(* Logix 5000 project; controller PlantaAutomatizacion vendor 1 type 14 code 156 rev 32.11; software revision 32.00 *)
// Planta de enesamblaje de patinetas electricas usando PLC Virtual.

TASK MainTask (continuous, watchdog 500 ms) : MainProgram

MODULES
   Local : vendor 1 type 14 code 156 (Compact 0, rev 32.11)
      Variador_141 : PowerFlex 525-EENET (Ethernet 10.203.3.141, rev 5.1, Output RPI 20 ms)
END_MODULES

VAR_GLOBAL   (* controller tags *)
   Banda1 : BOOL := 1;   // Motor de la banda 1
   Banda2 : BOOL := 1;   // Motor de la banda 2
   Banda3 : BOOL;   // Motor de la banda 3
   Banda4 : BOOL := 1;   // Motor de la Banda 4
   Banda5 : BOOL;   // Motor de la Banda 5
   Banda6 : BOOL;   // Motor de la banda 6
   Banda7 : BOOL;   // Motor de la Banda 7
   Google_Stp_Banda5 : BOOL;   // Stop con google assistant
   Google_Str_Banda5 : BOOL;   // Start Con Google Assistan
   RESET : BOOL;   // Reset del grafcet
   START : BOOL;   // Senal de inicio de la rutina
   StartBanda1 : BOOL := 1;   // Señal del sensor para activar Motor de la banda 1
   StartBanda2 : BOOL := 1;   // Señal del sensor para activar Motor de la banda 2
   StartBanda3 : BOOL;   // Señal del sensor para activar Motor de la banda 3
   StartBanda4 : BOOL := 1;   // Señal del sensor para activar Motor de la banda 4
   StartBanda5 : BOOL;   // Señal del sensor para activar Motor de la banda 5
   StartBanda6 : BOOL;   // Señal del sensor para activar Motor de la banda 6
   StartBanda7 : BOOL;   // Señal del sensor para activar Motor de la banda 7
   StopBanda1 : BOOL;   // Señal del sensor para desactivar Motor de la banda 1
   StopBanda2 : BOOL;   // Señal del sensor para desactivar Motor de la banda 2
   StopBanda3 : BOOL;   // Señal del sensor para desactivar Motor de la banda 3
   StopBanda4 : BOOL;   // Señal del sensor para desactivar Motor de la banda 4
   StopBanda5 : BOOL;   // Señal del sensor para desactivar Motor de la banda 5
   StopBanda6 : BOOL;   // Señal del sensor para desactivar Motor de la banda 6
   StopBanda7 : BOOL;   // Señal del sensor para desactivar Motor de la banda 7
END_VAR

PROGRAM MainProgram   (* main routine MainRoutine *)
VAR
   Action_000 : SFC_ACTION := (Status := 16#c020_0000, A := 1, Q := 1, PauseTimer := 1, Count := 1);   // Activar el Motor de la Banda
   Action_001 : SFC_ACTION := (Status := 16#0020_0000, PauseTimer := 1);
   Action_002 : SFC_ACTION := (Status := 16#c020_0000, A := 1, Q := 1, PauseTimer := 1, Count := 1);
   Action_003 : SFC_ACTION := (Status := 16#0020_0000, PauseTimer := 1);
   Action_004 : SFC_ACTION := (Status := 16#0020_0000, PauseTimer := 1);
   Action_005 : SFC_ACTION := (Status := 16#0020_0000, PauseTimer := 1);
   Action_006 : SFC_ACTION := (Status := 16#c020_0000, A := 1, Q := 1, PauseTimer := 1, Count := 1);
   Action_007 : SFC_ACTION := (Status := 16#0020_0000, PauseTimer := 1);
   Action_008 : SFC_ACTION := (Status := 16#0020_0000, PauseTimer := 1);
   Action_009 : SFC_ACTION := (Status := 16#0020_0000, PauseTimer := 1);
   Action_010 : SFC_ACTION := (Status := 16#0020_0000, PauseTimer := 1);
   Action_011 : SFC_ACTION := (Status := 16#0020_0000, PauseTimer := 1);
   Action_012 : SFC_ACTION := (Status := 16#0020_0000, PauseTimer := 1);
   Action_013 : SFC_ACTION := (Status := 16#0020_0000, PauseTimer := 1);
   Step_000 : SFC_STEP := (Status := 16#0820_0201, DN := 1, PauseTimer := 1, T := 400127, TMax := 400127, Count := 1);   // Paso Inicial
   Step_001 : SFC_STEP := (Status := 16#a820_0001, X := 1, SA := 1, DN := 1, PauseTimer := 1, T := 107426, TMax := 107426, Count := 1);   // Activar el Motor de la Banda
   Step_002 : SFC_STEP := (Status := 16#0020_0001, PauseTimer := 1);   // Detener el motor de la Banda
   Step_003 : SFC_STEP := (Status := 16#0820_0001, DN := 1, PauseTimer := 1, Count := 1);
   Step_004 : SFC_STEP := (Status := 16#a820_0001, X := 1, SA := 1, DN := 1, PauseTimer := 1, T := 107332, TMax := 107332, Count := 1);
   Step_005 : SFC_STEP := (Status := 16#0020_0001, PauseTimer := 1);
   Step_006 : SFC_STEP := (Status := 16#a820_0001, X := 1, SA := 1, DN := 1, PauseTimer := 1, T := 107361, TMax := 107361, Count := 1);
   Step_007 : SFC_STEP := (Status := 16#0020_0001, PauseTimer := 1);
   Step_008 : SFC_STEP := (Status := 16#0020_0001, PauseTimer := 1);
   Step_009 : SFC_STEP := (Status := 16#a820_0001, X := 1, SA := 1, DN := 1, PauseTimer := 1, T := 107408, TMax := 107408, Count := 1);
   Step_010 : SFC_STEP := (Status := 16#a820_0001, X := 1, SA := 1, DN := 1, PauseTimer := 1, T := 107437, TMax := 107437, Count := 1);
   Step_011 : SFC_STEP := (Status := 16#0020_0001, PauseTimer := 1);
   Step_012 : SFC_STEP := (Status := 16#a820_0001, X := 1, SA := 1, DN := 1, PauseTimer := 1, T := 107309, TMax := 107309, Count := 1);
   Step_013 : SFC_STEP := (Status := 16#0020_0001, PauseTimer := 1);
   Step_014 : SFC_STEP := (Status := 16#0020_0001, PauseTimer := 1);
   Step_015 : SFC_STEP := (Status := 16#0820_0001, DN := 1, PauseTimer := 1, Count := 1);   // Paso de paralelizado de las bandas
   Step_016 : SFC_STEP := (Status := 16#0020_0001, PauseTimer := 1);
   Step_017 : SFC_STEP := (Status := 16#0020_0001, PauseTimer := 1);
   Step_018 : SFC_STEP := (Status := 16#0820_0001, DN := 1, PauseTimer := 1, Count := 1);
   Step_019 : SFC_STEP := (Status := 16#a820_0001, X := 1, SA := 1, DN := 1, PauseTimer := 1, T := 107279, TMax := 107279, Count := 1);
   Step_020 : SFC_STEP := (Status := 16#0020_0001, PauseTimer := 1);
   Step_021 : SFC_STEP := (Status := 16#0020_0001, PauseTimer := 1);
   Tran_000 : BOOL := 1;   // Sensor de banda 1 indicando que hay un Objeto
   Tran_001 : BOOL;   // Sensor de parada, indicando qeu el objeto llego a su destino
   Tran_002 : BOOL;   // Cuando El objeto ya halla sido recogido Y otro objeto se encuentre al incio
   Tran_003 : BOOL := 1;
   Tran_004 : BOOL;
   Tran_005 : BOOL;
   Tran_006 : BOOL;
   Tran_007 : BOOL;
   Tran_008 : BOOL := 1;
   Tran_009 : BOOL := 1;
   Tran_010 : BOOL;
   Tran_011 : BOOL;
   Tran_012 : BOOL;
   Tran_013 : BOOL := 1;
   Tran_014 : BOOL;
   Tran_015 : BOOL;
   Tran_016 : BOOL := 1;
   Tran_017 : BOOL;
   Tran_018 : BOOL;
   Tran_019 : BOOL := 1;
   Tran_020 : BOOL;
   Tran_022 : BOOL := 1;   // START para empezar la logica grafcet
END_VAR

ROUTINE GrafcetBandas   (* sequential function chart *)
// Logica secuencial para el movimiento de las bandas
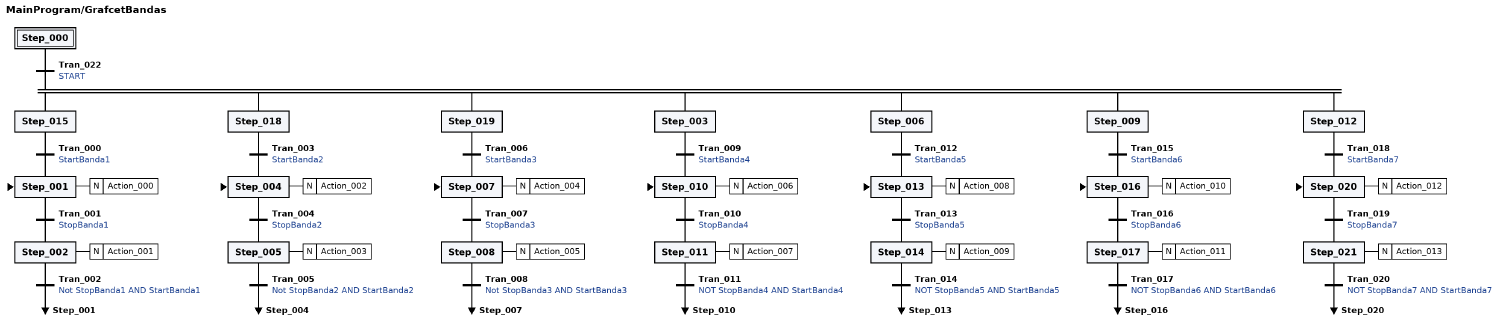
   // BANDA 1
   // BANDA 2
   // BANDA 3
   // BANDA 4
   // BANDA 5
   // BANDA 6
   // BANDA 7
   INITIAL_STEP Step_000:
   END_STEP
   TRANSITION Tran_022 FROM Step_000 TO (Step_018, Step_019, Step_015, Step_003, Step_006, Step_009, Step_012)
      := START
   END_TRANSITION
   STEP Step_015:
   END_STEP
   STEP Step_018:
   END_STEP
   STEP Step_019:
   END_STEP
   STEP Step_003:
   END_STEP
   STEP Step_006:
   END_STEP
   STEP Step_009:
   END_STEP
   STEP Step_012:
   END_STEP
   TRANSITION Tran_015 FROM Step_009 TO Step_016
      := StartBanda6
   END_TRANSITION
   TRANSITION Tran_018 FROM Step_012 TO Step_020
      := StartBanda7
   END_TRANSITION
   TRANSITION Tran_000 FROM Step_015 TO Step_001
      := StartBanda1
   END_TRANSITION
   TRANSITION Tran_003 FROM Step_018 TO Step_004
      := StartBanda2
   END_TRANSITION
   TRANSITION Tran_006 FROM Step_019 TO Step_007
      := StartBanda3
   END_TRANSITION
   TRANSITION Tran_009 FROM Step_003 TO Step_010
      := StartBanda4
   END_TRANSITION
   TRANSITION Tran_012 FROM Step_006 TO Step_013
      := StartBanda5
   END_TRANSITION
   STEP Step_016:
      ACTION Action_010 (N):
         Banda6:=1;
      END_ACTION
   END_STEP
   STEP Step_020:
      ACTION Action_012 (N):
         Banda7:=1;
      END_ACTION
   END_STEP
   STEP Step_001:
      ACTION Action_000 (N):
         Banda1:=1;
      END_ACTION
   END_STEP
   STEP Step_004:
      ACTION Action_002 (N):
         Banda2:=1;
      END_ACTION
   END_STEP
   STEP Step_007:
      ACTION Action_004 (N):
         Banda3:=1;
      END_ACTION
   END_STEP
   STEP Step_010:
      ACTION Action_006 (N):
         Banda4:=1;
      END_ACTION
   END_STEP
   STEP Step_013:
      ACTION Action_008 (N):
         Banda5:=1;
      END_ACTION
   END_STEP
   TRANSITION Tran_016 FROM Step_016 TO Step_017
      := StopBanda6
   END_TRANSITION
   TRANSITION Tran_019 FROM Step_020 TO Step_021
      := StopBanda7
   END_TRANSITION
   TRANSITION Tran_001 FROM Step_001 TO Step_002
      := StopBanda1
   END_TRANSITION
   TRANSITION Tran_004 FROM Step_004 TO Step_005
      := StopBanda2
   END_TRANSITION
   TRANSITION Tran_007 FROM Step_007 TO Step_008
      := StopBanda3
   END_TRANSITION
   TRANSITION Tran_010 FROM Step_010 TO Step_011
      := StopBanda4
   END_TRANSITION
   TRANSITION Tran_013 FROM Step_013 TO Step_014
      := StopBanda5
   END_TRANSITION
   STEP Step_017:
      ACTION Action_011 (N):
         Banda6:=0;
      END_ACTION
   END_STEP
   STEP Step_021:
      ACTION Action_013 (N):
         Banda7:=0;
      END_ACTION
   END_STEP
   STEP Step_002:
      ACTION Action_001 (N):
         Banda1:=0;
      END_ACTION
   END_STEP
   STEP Step_005:
      ACTION Action_003 (N):
         Banda2:=0;
      END_ACTION
   END_STEP
   STEP Step_008:
      ACTION Action_005 (N):
         Banda3:=0;
      END_ACTION
   END_STEP
   STEP Step_011:
      ACTION Action_007 (N):
         Banda4:=0;
      END_ACTION
   END_STEP
   STEP Step_014:
      ACTION Action_009 (N):
         Banda5:=0;
      END_ACTION
   END_STEP
   TRANSITION Tran_002 FROM Step_002 TO Step_001
      := Not StopBanda1
         AND StartBanda1
   END_TRANSITION
   TRANSITION Tran_005 FROM Step_005 TO Step_004
      := Not StopBanda2
         AND StartBanda2
   END_TRANSITION
   TRANSITION Tran_008 FROM Step_008 TO Step_007
      := Not StopBanda3
         AND StartBanda3
   END_TRANSITION
   TRANSITION Tran_011 FROM Step_011 TO Step_010
      := NOT StopBanda4
         AND StartBanda4
   END_TRANSITION
   TRANSITION Tran_014 FROM Step_014 TO Step_013
      := NOT StopBanda5
         AND StartBanda5
   END_TRANSITION
   TRANSITION Tran_017 FROM Step_017 TO Step_016
      := NOT StopBanda6
         AND StartBanda6
   END_TRANSITION
   TRANSITION Tran_020 FROM Step_021 TO Step_020
      := NOT StopBanda7
         AND StartBanda7
   END_TRANSITION
END_ROUTINE

ROUTINE MainRoutine   (* ladder *)
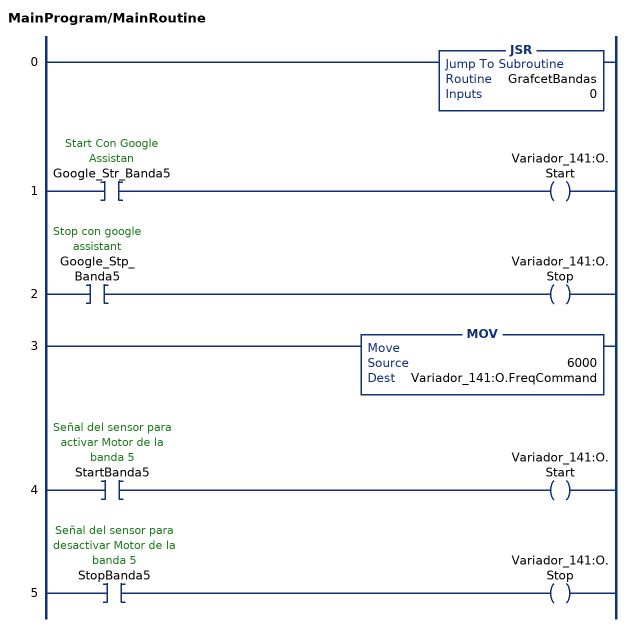
   0: JSR(GrafcetBandas,0);
   1: XIC(Google_Str_Banda5)OTE(Variador_141:O.Start);
   2: XIC(Google_Stp_Banda5)OTE(Variador_141:O.Stop);
   3: MOV(6000,Variador_141:O.FreqCommand);
   4: XIC(StartBanda5)OTE(Variador_141:O.Start);
   5: XIC(StopBanda5)OTE(Variador_141:O.Stop);
END_ROUTINE
END_PROGRAM
